ABB RobotStudio station: LearningSolution_20201008-232713.rsstn

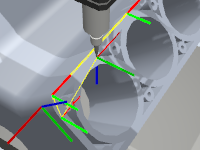
Station LearningSolution (saved by RobotStudio 20.2.9116.0)
Controller LearningController1
  mechanical unit ROB_1: IRB4600_20_250_C_01, 6 joints, base frame (0, 0, 0) mm
Layout (positions relative to the parent item):
  - IRB4600_20_250_C_01 [mechanism, from Robots\IRB4600_20_250_C_G_01.rslib] at (0, 0, 0) mm; joint values [0.2011, 0.3306, 0.3286, -0.4517, 0.2856, 0.5949] (rad or m)
  - MyTool [mechanism, from Training Objects\myTool.rslib] at (1630.24, 321.62, 848.42) mm, rotated rx -180 ry 38 rz 180 deg
  - Table [part] at (1374.27, -200, 0) mm
  - Engine Block [part] at (1630.97, 175, 400) mm, rotated rx 90.36 ry 0 rz 0 deg
Attachment: MyTool is attached to IRB4600_20_250_C_01 / Link6
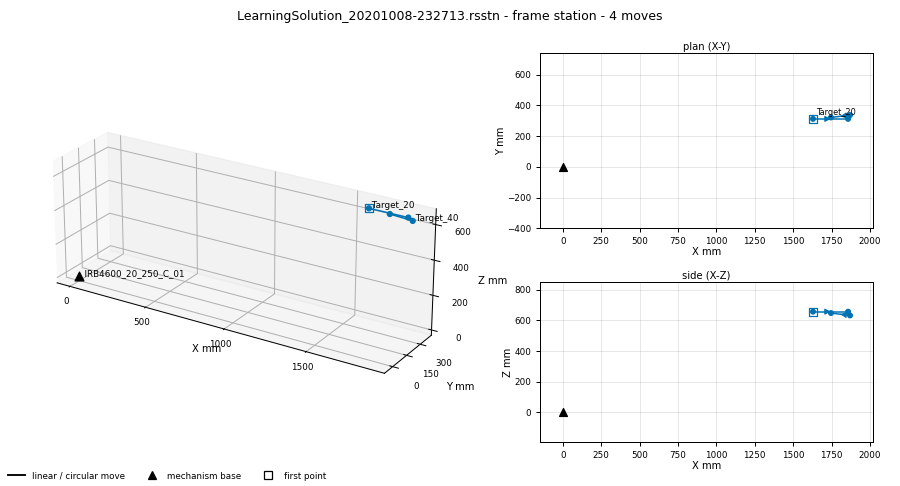
[picture p0: tool path of LearningSolution_20201008-232713.rsstn in frame station, 4 of 4 moves have a stored position in this frame; points joined in program order, loops and branches not executed]
Targets, tools, work objects and paths stored in the station, written as RAPID:
! task T_ROB1
MODULE CalibData
  PERS tooldata MyTool:=[TRUE,[[31.792631019,0,229.638935148],[0.945518576,0,0.325568154,0]],[1,[0,0,1],[1,0,0,0],0,0,0]];
  TASK PERS wobjdata wobj_engine:=[FALSE,TRUE,"",[[1883.468402126,312.582,656.808],[0.925076886,-0.379779878,0,0]],[[0,0,0],[1,0,0,0]]];
ENDMODULE

! task T_ROB1
MODULE Module1
  CONST robtarget Target_20:=[[-254,0,0],[0,0,0.925076886,0.379779878],[0,0,0,0],[9E+09,9E+09,9E+09,9E+09,9E+09,9E+09]];
  CONST robtarget Target_30:=[[-25.4,0,0],[0,0,0.925076886,0.379779878],[0,-1,0,0],[9E+09,9E+09,9E+09,9E+09,9E+09,9E+09]];
  CONST robtarget Target_40:=[[-12.7,35.066821939,-0.000360378],[0,0,0.925076886,0.379779878],[0,-1,0,0],[9E+09,9E+09,9E+09,9E+09,9E+09,9E+09]];
  CONST robtarget Target_60:=[[-136.901402126,12.699884711,-0.000577776],[0,0,0.925076886,0.379779878],[0,-1,0,0],[9E+09,9E+09,9E+09,9E+09,9E+09,9E+09]];
  PROC Path_10()
    MoveJ Target_20,v50,z5,MyTool\WObj:=wobj_engine;
    MoveL Target_30,v50,z5,MyTool\WObj:=wobj_engine;
    MoveL Target_40,v50,z5,MyTool\WObj:=wobj_engine;
    MoveL Target_60,v50,z5,MyTool\WObj:=wobj_engine;
  ENDPROC
  PROC main()
    Path_10;
  ENDPROC
ENDMODULE

